// SIMATIC S7-200 SMART project (STEP 7-Micro/WIN SMART), CPU SR40

SYMBOL_TABLE USR1
右起动              I0.0
左起动              I0.1
停车               I0.2
左限位              I0.3
右限位              I0.4
过载               I0.5
右行               Q0.0
左行               Q0.1
END_SYMBOL_TABLE

SYMBOL_TABLE 用户定义2
rejidianqi
tingche
youqidong
youshuchu
youxianwei
zuoqidong
zuoshuchu
zuoxianwei
END_SYMBOL_TABLE

ORGANIZATION_BLOCK MAIN:OB1
TITLE=程序注释
BEGIN
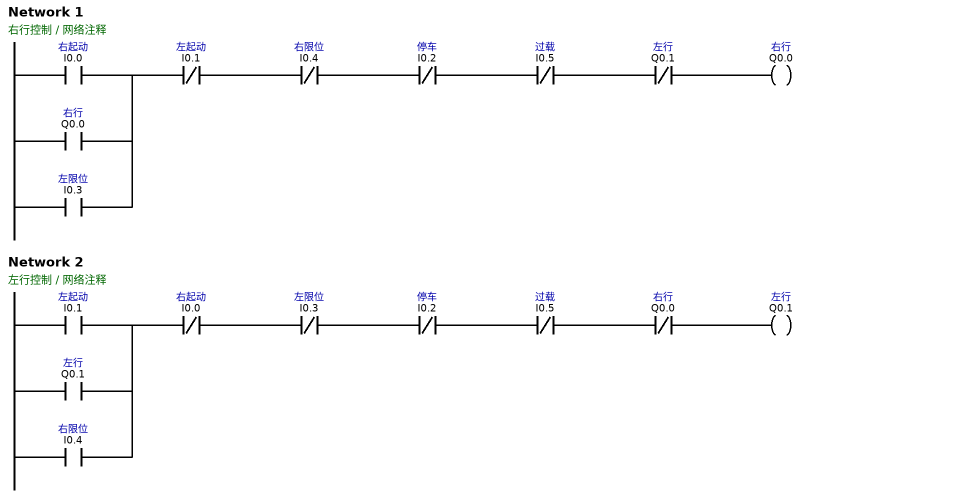
Network 1
// 右行控制
// 网络注释
// (network saved uncompiled; LAD cells follow)
// row 0: c0 -| |- 右起动:I0.0 v  c1 -|/|- 左起动:I0.1  c2 -|/|- 右限位:I0.4  c3 -|/|- 停车:I0.2  c4 -|/|- 过载:I0.5  c5 -|/|- 左行:Q0.1  c6 -( ) 右行:Q0.0
// row 1: c0 -| |- 右行:Q0.0 ^v
// row 2: c0 -| |- 左限位:I0.3 ^
Network 2
// 左行控制
// 网络注释
// (network saved uncompiled; LAD cells follow)
// row 0: c0 -| |- 左起动:I0.1 v  c1 -|/|- 右起动:I0.0  c2 -|/|- 左限位:I0.3  c3 -|/|- 停车:I0.2  c4 -|/|- 过载:I0.5  c5 -|/|- 右行:Q0.0  c6 -( ) 左行:Q0.1
// row 1: c0 -| |- 左行:Q0.1 ^v
// row 2: c0 -| |- 右限位:I0.4 ^
END_ORGANIZATION_BLOCK
